// TIA Portal V18 export
TYPE "RCS_SysStatus_V1"
   STRUCT
      ControlOn : Bool;   // System Control On Status
      ControlOff : Bool;   // System Control Off Status
      Run : Bool;   // Delay from control on and E-stopOK for 3-5 second
      EStopOK : Bool;   // all Estop Button released and be reset
      EnableAlarm : Bool;   // Station can activate Alarm
      Error : Bool;   // Station in Alarm/Error status
      FixtureOK : Bool;
      ChangeOverOK : Bool;
      AllDeviceReady : Bool;   // All peripheral device comunication ok and in ready status
      Ready : Bool;   // Station in AutoMode and all Status OK, ready for AutoRuning
      CanStart : Bool;
      Home : Bool;   // Station at Home position
      WaitMaterial : Bool;
      LightCurtainOK : Bool;   // All Light Curtain OK and be reset
      SaftyDoorOK : Bool;   // All Safty Door closed and Locked, be reset
      MainPressureOK : Bool;   // All Main air source PressureOK
      ModeSV : Int;   // 1Manual,2Auto,3Step, 4OneCycle
      ModePV : Int;   // 0NA,1Manual, 2Auto, 3Step, 4OneCycle, 5Runn, 6Error
      FinishProduct : DInt;   // 0NA,1=OK,other=NG
   END_STRUCT;
END_TYPE
